FUNCTION_BLOCK ArrayCumulative (* Basic FB with empty ECC *)
  (* Standard: 61499-2; Function: Summing all the components of array input *)
  (* Version 1.0, 2020-07-16, Candra Wardaya, UGM *)
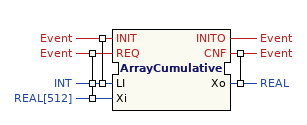
  EVENT_INPUT
    INIT WITH LI; (* Initialization In *)
    REQ WITH LI, Xi; (* Execution Request *)
  END_EVENT
  EVENT_OUTPUT
    INITO; (* Initialization Out *)
    CNF WITH Xo; (* Confirmation of Execution *)
  END_EVENT
  VAR_INPUT
    LI : INT; (* Array Length *)
    Xi : ARRAY [0..511] OF REAL; (* Array Input *)
  END_VAR
  VAR_OUTPUT
    Xo : REAL; (* Output real, cumulative *)
  END_VAR
  VAR
    i : INT; (* Internal Variable *)
    val : REAL; (* Internal Variable *)
  END_VAR
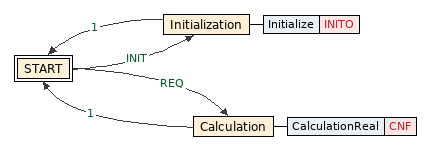
  EC_STATES
    START; (* Initial State *)
    Initialization : Initialize -> INITO;
    Calculation : CalculationReal -> CNF;
  END_STATES
  EC_TRANSITIONS
    START TO Initialization := INIT;
    Initialization TO START := 1;
    START TO Calculation := REQ;
    Calculation TO START := 1;
  END_TRANSITIONS
  ALGORITHM CalculationReal IN ST: (* New Algorithm *)
val :=0;
for i:=0 to LI-1 do
	val := val + Xi[i];
end_for;
Xo := val;
  END_ALGORITHM
  ALGORITHM Initialize IN ST: (* New Algorithm *)

  END_ALGORITHM
END_FUNCTION_BLOCK
